# B&R Automation Studio project FileBrowse
Automation Studio 4.12.2.93; technology packages: mapp 5.24.1, mappView 5.24.2

## Configuration APC2200

CPU 5PPC2200.AL14-000, AutomationRuntime H4.93, Build 4.1.2, Vc V4.72.6

### Task classes (Cpu.sw)
```
Cyclic#1:
  Program <- Program.prg
Libraries: operator, runtime, astime, AsIecCon, FileBrowse, MpFile, FileIO, MpBase, AsBrStr, standard
```

### Hardware
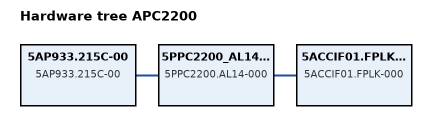
```
5ACCIF01.FPLK-000 : 5ACCIF01.FPLK-000 v1.7.1.0  [SL -> 5PPC2200_AL14_000.SL1]
5AP933.215C-00 : 5AP933.215C-00 v2.0.0.0
5PPC2200_AL14_000 : 5PPC2200.AL14-000 v2.0.6.0  [SY -> 5AP933.215C-00.SY1]
  Connector IF3:
    AssignedOperatingSystem = ARemb
    ActivateDevice = 1
    ActivateSnmp = 2
  Connector IF4:
    AssignedOperatingSystem = ARemb
    ActivateDevice = 1
    ActivateSnmp = 2
  Connector IF7:
    OperatingSystem = ARemb
    ActivateDevice = 1
  Connector IF5:
    AssignedOperatingSystem = ARemb
  Connector IF6:
    AssignedOperatingSystem = ARemb
  ConfigurationID = FileBrowse_APC2200
  UserPartitionSize = 20
  UserRamDevice = PCI.1.PPC21xx.SRAM
  UserRamSize = 5000
  EnableUsbRemoteInstall = 1
  FileDevice1
  FileDeviceName1 = USER
  FileDevicePath1 = USER_PATH
  ActivateOpcUa = 1
  OpcUaPort = 4841
  OpcUaInformationModels_PV_Version = 1
  ActivateHypervisor = 1
```

## Configuration ArSim

CPU PC_any, AutomationRuntime K4.93, Build 4.1.2, Vc V4.72.6

### Task classes (Cpu.sw)
```
Cyclic#4:
  Program <- Program.prg
Libraries: FileBrowse, MpFile, FileIO, MpBase, runtime, AsBrStr, standard
```

### Hardware
```
PC : PC_any v1.1.1.0 (OrderNumber=PC)
  ConfigurationID = FileBrowse_ArSim
  FileDevice1
  FileDeviceName1 = USER
  FileDevicePath1 = USER_PATH
  ActivateOpcUa = 1
  OpcUaInformationModels_PV_Version = 1
```

## Logical view

Binary libraries used (declarations not repeated): operator, runtime, astime, AsIecCon, MpFile, FileIO, MpBase, AsBrStr, standard

### Library Logical/Libraries/FileBrowse (IEC)
Depends on: standard, AsBrStr, MpFile, FileIO, MpBase

#### Constants.var - Exported constants
```iecst
VAR CONSTANT
	STRINGCMP_NO_DIFF : USINT := 0;
END_VAR
```

#### FileBrowse.fun - Exported functions and function blocks
```iecst
FUNCTION_BLOCK FileBrowseMV
	VAR_INPUT
		NetworkConnectionOK : BOOL; (*Allows selection of Network files (DevLink) if set up.*)
		FileDevices : ARRAY[0..2] OF STRING[40]; (*Files devices are listed in order, Local user partition, Network, USB*)
		MpLink : UDINT; (*Address of mappFileManagerUI*)
		USB_Detected : BOOL; (*Allows selection of USB files if setup*)
	END_VAR
	VAR_OUTPUT
		FilePath : STRING[200]; (*Path to chosen file*)
	END_VAR
	VAR_INPUT
		ShowDialog : BOOL; (*True when filebrowsing is occuring. This was tied to a pop up in mapp view.*)
	END_VAR
	VAR
		Index : UINT; (*Index of focused file in current directory*)
		CurrentPage : USINT; (*Page number withing directory*)
		Filter : STRING[40]; (*Text that is being looked for*)
		FilterInput : BOOL; (*Indication that filter has been applied*)
		DataProvider : ARRAY[0..49] OF STRING[100]; (*Output text to mappview to be displayed in listbox*)
		Open : BOOL; (*Command to select the currently focused file and update the FilePath*)
		MaxPages : USINT; (*Total number of pages based on number of files in current directory*)
		temp : STRING[200]; (*Temp string*)
		ToggleNetwork : BOOL; (*Toggle status of network button*)
		ToggleUSB : BOOL; (*Toggle status of USB button*)
		ToggleLocal : BOOL; (*Toggle status of Local button (User partition)*)
		TotalIndex : UDINT; (*Total number of file and folders found within current directory*)
		PreviousDevice : UINT; (*Last selected device*)
		EnteredFolderCnt : USINT; (*Keeps track of how many levels deep within a folder user has gone, used for folder back button visibility*)
		FolderUp : BOOL; (*Command to exit out of current folder, going up a level*)
		WaitForRefresh : BOOL; (*Flag for refreshing list*)
		TON_Refresh : TON; (*Timer for refreshing list*)
		Close : BOOL;
		ListClicked : BOOL; (*Indicates that user has clicked on the list *)
		PreviousIndex : UINT; (*Keep tracks of last focused index*)
		TempStringArrayIndex : UINT;
		i : UINT;
		ShowFolderBackBtn : BOOL; (*Visibility of folder back button*)
		MpFileManagerUI_FB : MpFileManagerUI;
		UIconnect : MpFileManagerUIConnectType;
		UIsetup : MpFileManagerUISetupType;
		zzEdge00000 : BOOL;
		zzEdge00001 : BOOL;
		zzEdge00002 : BOOL;
		zzEdge00003 : BOOL;
	END_VAR
END_FUNCTION_BLOCK
```

#### FileBrowseMV.st
```iecst
(* Controls compound widget to interact with mpFileUI to display a file browser. *)
FUNCTION_BLOCK FileBrowseMV
	UIconnect.DeviceList.DeviceNames[0]	:= FileDevices[0];
	UIconnect.DeviceList.DeviceNames[1]	:= FileDevices[1];
	UIconnect.DeviceList.DeviceNames[2]	:= FileDevices[2];

	MpFileManagerUI_FB.MpLink 		:= MpLink;
	MpFileManagerUI_FB.Enable		:= TRUE;
	MpFileManagerUI_FB.ErrorReset;
	MpFileManagerUI_FB.UIConnect	:= ADR(UIconnect);
	MpFileManagerUI_FB.UISetup		:= UIsetup;
	//Timer delay on refresh. FB needs to run an indeterminate amount of cycles before a refresh
	IF TON_Refresh.Q THEN
		UIconnect.File.Refresh	:= TRUE;
		WaitForRefresh		:= FALSE;
		Index				:= 0;
		TotalIndex			:= 0;
	END_IF

	IF EDGEPOS(ShowDialog) THEN
		UIconnect.File.Refresh			:= TRUE;
	END_IF

	//Go to local if connection lost
	IF ToggleNetwork AND NOT(NetworkConnectionOK) THEN
		ToggleLocal	:= TRUE;
	ELSIF ToggleUSB AND NOT(USB_Detected) THEN
		ToggleLocal	:= TRUE;
	END_IF
	//Refresh when changing devices
	IF PreviousDevice <> UIconnect.DeviceList.SelectedIndex THEN
		WaitForRefresh					:= TRUE;
		PreviousDevice					:= UIconnect.DeviceList.SelectedIndex;
	END_IF
	ShowFolderBackBtn	:= (EnteredFolderCnt > 0);
	// Only runs while  selection dialog is open
	IF ShowDialog THEN
		//Count number of total pages
		MaxPages 					:= UDINT_TO_USINT((UIconnect.File.PathInfo.FileCount + UIconnect.File.PathInfo.FolderCount) / UIsetup.FileListSize);
		IF (UIconnect.File.PathInfo.FileCount + UIconnect.File.PathInfo.FolderCount) > (UIsetup.FileListSize * MaxPages) THEN
			MaxPages					:= MaxPages + 1;
		END_IF
		IF MaxPages < 1 THEN
			MaxPages	:= 1;
		END_IF

		//Resets all values when changing devices
		IF EDGEPOS(ToggleNetwork) THEN
			Index							:= 0;
			TotalIndex						:= 0;
			EnteredFolderCnt					:= 0;
			ToggleUSB						:= FALSE;
			ToggleLocal						:= FALSE;
			UIconnect.DeviceList.SelectedIndex 	:= 1;
		END_IF
		IF EDGEPOS(ToggleLocal) THEN
			Index							:= 0;
			TotalIndex						:= 0;
			EnteredFolderCnt					:= 0;
			ToggleUSB						:= FALSE;
			ToggleNetwork					:= FALSE;
			UIconnect.DeviceList.SelectedIndex 	:= 0;
		END_IF
		IF EDGEPOS(ToggleUSB) THEN
			Index							:= 0;
			TotalIndex						:= 0;
			EnteredFolderCnt					:= 0;
			ToggleLocal						:= FALSE;
			ToggleNetwork					:= FALSE;
			UIconnect.DeviceList.SelectedIndex 	:= 2;
		END_IF
		// Goes back to Local file device if USB connection is lost
		IF UIconnect.DeviceList.SelectedIndex = 2 AND NOT(USB_Detected) THEN
			ToggleLocal		:= TRUE;
		END_IF
		//Adjusts filter to not be exact
		IF FilterInput THEN
			brsstrcpy(ADR(UIconnect.File.Filter),ADR('*'));
			brsstrcat(ADR(UIconnect.File.Filter),ADR(Filter));
			brsstrcat(ADR(UIconnect.File.Filter),ADR('*'));
			WaitForRefresh		:= TRUE;
			FilterInput				:= FALSE;
		END_IF
		//Updates the  list
		brsmemset(ADR(DataProvider),0,SIZEOF(DataProvider));
		FOR i:= 0 TO UIsetup.FileListSize BY 1 DO
			IF brsstrcmp(ADR(UIconnect.File.List.Items[i].Name),ADR('')) <> STRINGCMP_NO_DIFF THEN
				brsmemset(ADR(DataProvider[i]),0,SIZEOF(DataProvider[i]));
				brsstrcat(ADR(DataProvider[i]),ADR('{"value":"'));
				brsitoa(i,ADR(TempStringArrayIndex));
				brsstrcat(ADR(DataProvider[i]),ADR(TempStringArrayIndex));
				brsstrcat(ADR(DataProvider[i]),ADR('","text":"'));
				brsstrcat(ADR(DataProvider[i]),ADR(UIconnect.File.List.Items[i].Name));
				brsstrcat(ADR(DataProvider[i]),ADR('"}'));
			END_IF
		END_FOR
		//Updates TotalIndex and makes sure correct  is selected when user touchs the list
		IF ListClicked THEN
			IF Index < PreviousIndex THEN
				TotalIndex	:= TotalIndex - (PreviousIndex - Index);
			ELSE
				TotalIndex	:= TotalIndex + (Index - PreviousIndex);
			END_IF
			UIconnect.File.List.Items[Index].IsSelected	:= TRUE;
			ListClicked	:= FALSE;
		END_IF
		// index calculations based on actions taken and current position within list
		IF UIconnect.File.List.StepUp THEN
			IF Index > 0 THEN
				Index		:= Index - 1;
			END_IF
			IF TotalIndex > 0 THEN
				TotalIndex	:= TotalIndex - 1;
			END_IF
		ELSIF UIconnect.File.List.StepDown THEN
			IF Index < (UIsetup.FileListSize - 1) AND Index < (UIconnect.File.PathInfo.FileCount + UIconnect.File.PathInfo.FolderCount - 1)  THEN
				Index		:= Index + 1;
			END_IF
			IF TotalIndex < (UIconnect.File.PathInfo.FileCount + UIconnect.File.PathInfo.FolderCount - 1) THEN
				TotalIndex	:= TotalIndex + 1;
			END_IF
		ELSIF UIconnect.File.List.PageUp THEN
			IF Index > 0 THEN
				TotalIndex	:= TotalIndex - Index;
				Index		:= 0;
			ELSIF CurrentPage > 1 THEN
				TotalIndex	:= TotalIndex - (UIsetup.FileListSize - 1);
			ELSE
				TotalIndex	:= 0;
			END_IF
		ELSIF UIconnect.File.List.PageDown THEN
			IF Index < (UIsetup.FileListSize - 1) AND Index < (UIconnect.File.PathInfo.FileCount + UIconnect.File.PathInfo.FolderCount - 1)  THEN
				TotalIndex	:= TotalIndex + MIN(UDINT_TO_UINT((UIconnect.File.PathInfo.FileCount + UIconnect.File.PathInfo.FolderCount - 1)),(UIsetup.FileListSize - 1 - Index));
				Index		:= MIN(UDINT_TO_UINT((UIconnect.File.PathInfo.FileCount + UIconnect.File.PathInfo.FolderCount - 1)),(UIsetup.FileListSize - 1));
			ELSIF UIconnect.File.List.RangeStart > 0 THEN
				TotalIndex	:= MIN((TotalIndex + (UIsetup.FileListSize - 1)),(UIconnect.File.PathInfo.FileCount + UIconnect.File.PathInfo.FolderCount - 1));
			END_IF
		END_IF
		// Current  page
		IF TotalIndex > 0 THEN
			CurrentPage	:= UDINT_TO_USINT(TotalIndex / UIsetup.FileListSize) + 1;
		ELSE
			CurrentPage	:= 1;
		END_IF
		IF CurrentPage = 1 THEN
			// Weird timing issue sometimes causes TotalIndex to not update properly, this will hopefully minimize the chances of that happening
			TotalIndex		:= Index;
		END_IF
		PreviousIndex	:= Index;
	END_IF

	IF Open THEN
		IF UIconnect.File.List.Items[Index].IsFolder THEN
			UIconnect.File.EnterFolder	:= TRUE;
			WaitForRefresh			:= TRUE;
			EnteredFolderCnt			:= EnteredFolderCnt + 1;
		ELSE
			brsstrcpy(ADR(FilePath),ADR(''));
			// assemble in format that MpCnc wants (FileDev:Path/File)
			brsstrcpy(ADR(temp), ADR(UIconnect.DeviceList.DeviceNames[UIconnect.DeviceList.SelectedIndex]));
			brsstrcat(ADR(temp), ADR(':'));
			IF brsstrcmp(ADR(UIconnect.File.PathInfo.CurrentDir),ADR('')) <> STRINGCMP_NO_DIFF THEN
				brsstrcat(ADR(temp), ADR(UIconnect.File.PathInfo.CurrentDir));
				brsstrcat(ADR(temp), ADR('/'));
				brsstrcpy(ADR(FilePath),ADR(UIconnect.File.PathInfo.CurrentDir));
				brsstrcat(ADR(FilePath), ADR('/'));
			END_IF
			brsstrcat(ADR(temp), ADR(UIconnect.File.List.Items[Index].Name));
			brsstrcat(ADR(FilePath),ADR(UIconnect.File.List.Items[Index].Name));
			Close	:= TRUE;
		END_IF
		Open		:= FALSE;
	END_IF

	//Allows user to move up a directory
	IF EnteredFolderCnt > 0 AND FolderUp THEN
		UIconnect.File.FolderUp 	:= TRUE;
		WaitForRefresh				:= TRUE;
		FolderUp					:= FALSE;
		EnteredFolderCnt			:= EnteredFolderCnt - 1;
	END_IF
	//Resets counts
	IF NOT(ShowDialog) AND NOT(Open)THEN
		TotalIndex				:= 0;
		Index					:= 0;
		WaitForRefresh			:= 0;
		brsstrcpy(ADR(Filter),ADR(''));
		CurrentPage				:= 1;
		Close					:= 0;
		brsstrcpy(ADR(UIconnect.File.Filter),ADR(''));
	END_IF
	TON_Refresh(IN := WaitForRefresh, PT := T#700ms);
	MpFileManagerUI_FB();

END_FUNCTION_BLOCK
```

### Program Logical/Program

#### Variables.var
```iecst
VAR
	FileBrowseMV_0 : FileBrowseMV;
	NetworkOK : BOOL;
	USB_OK : BOOL;
	ShowDialog : BOOL;
END_VAR
```

#### Main.st
```iecst
PROGRAM _INIT
	(* Insert code here *)

END_PROGRAM

PROGRAM _CYCLIC
	(* Insert code here *)
	FileBrowseMV_0.FileDevices[0] 	:= 'USER';
	FileBrowseMV_0.NetworkConnectionOK	:= NetworkOK;
	FileBrowseMV_0.MpLink				:= ADR(gFileManagerUI);
	FileBrowseMV_0.USB_Detected			:= USB_OK;
	FileBrowseMV_0.ShowDialog			:= ShowDialog;
	FileBrowseMV_0();

END_PROGRAM

PROGRAM _EXIT
	(* Insert code here *)

END_PROGRAM
```

Listed in the project but not available here: Logical/Libraries/FileBrowse/Types.typ
